// SIMATIC S7-200 project (STEP 7-Micro/WIN), CPU 221 REL 01.10

ORGANIZATION_BLOCK MAIN:OB1
TITLE=
BEGIN
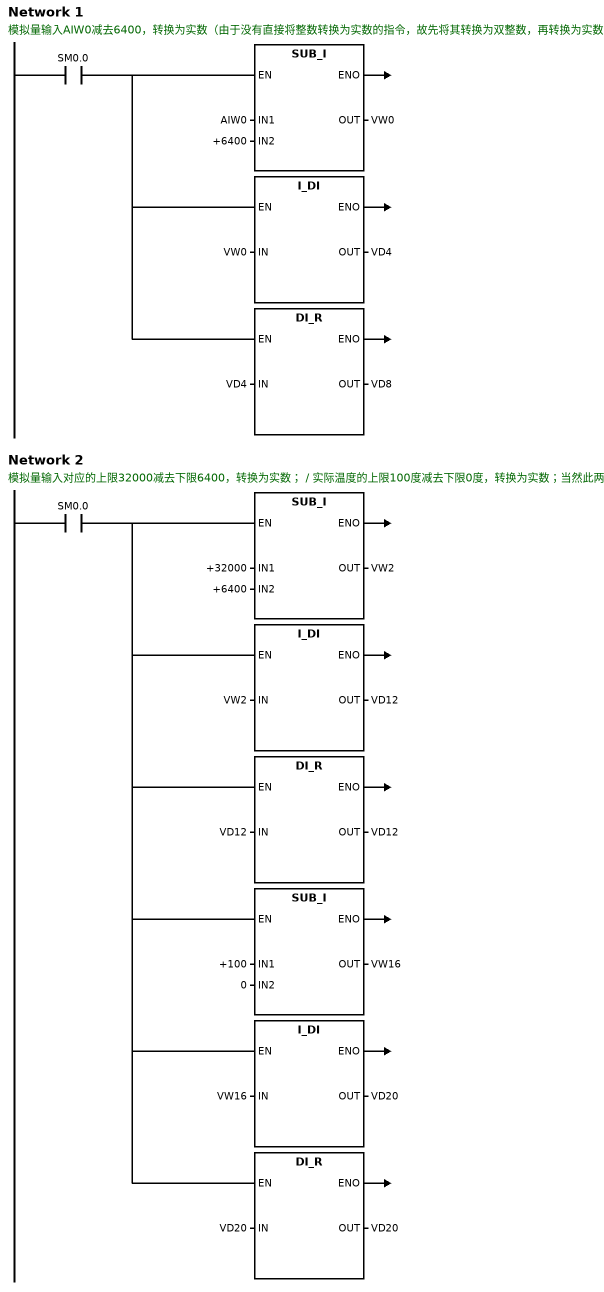
Network 1
// 模拟量输入AIW0减去6400，转换为实数（由于没有直接将整数转换为实数的指令，故先将其转换为双整数，再转换为实数）
LD     SM0.0
MOVW   AIW0, VW0
-I     +6400, VW0
ITD    VW0, VD4
DTR    VD4, VD8
Network 2
// 模拟量输入对应的上限32000减去下限6400，转换为实数；
// 实际温度的上限100度减去下限0度，转换为实数；当然此两步转换可以直接计算出来，这里主要想演示指令的使用
// (network saved uncompiled; LAD cells follow)
// row 0: c0 -| |- SM0.0 v  c1 --  c2 [SUB_I EN:=power@row0, IN1:=+32000, IN2:=+6400, ENO=>power, OUT=>VW2]  c3 ->
// row 1: c0 ^v  c2 [box]
// row 2: c0 ^v  c1 --  c2 [I_DI EN:=power@row2, IN:=VW2, ENO=>power, OUT=>VD12]  c3 ->
// row 3: c0 ^v  c2 [box]
// row 4: c0 ^v  c1 --  c2 [DI_R EN:=power@row4, IN:=VD12, ENO=>power, OUT=>VD12]  c3 ->
// row 5: c0 ^v  c2 [box]
// row 6: c0 ^v  c1 --  c2 [SUB_I EN:=power@row6, IN1:=+100, IN2:=0, ENO=>power, OUT=>VW16]  c3 ->
// row 7: c0 ^v  c2 [box]
// row 8: c0 ^v  c1 --  c2 [I_DI EN:=power@row8, IN:=VW16, ENO=>power, OUT=>VD20]  c3 ->
// row 9: c0 ^v  c2 [box]
// row 10: c0 ^  c1 --  c2 [DI_R EN:=power@row10, IN:=VD20, ENO=>power, OUT=>VD20]  c3 ->
// row 11: c2 [box]
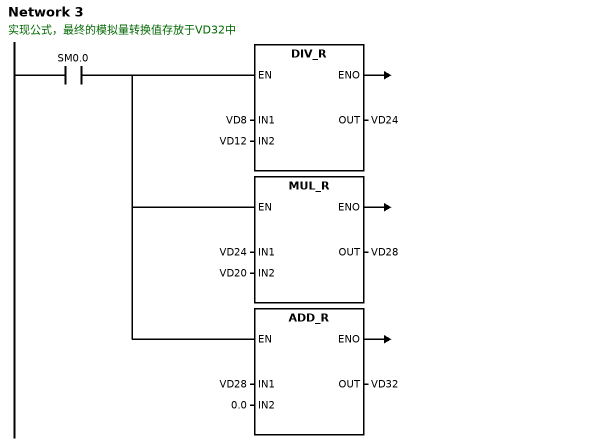
Network 3
// 实现公式，最终的模拟量转换值存放于VD32中
LD     SM0.0
MOVR   VD8, VD24
/R     VD12, VD24
MOVR   VD24, VD28
*R     VD20, VD28
MOVR   VD28, VD32
+R     0.0, VD32
END_ORGANIZATION_BLOCK
